// TIA Portal V20 export
TYPE "LConSMC_typePIDController"
// stored: Access Published
   STRUCT
      In { S7_SetPoint := 'True'} : "LConSMC_typePIDControllerIn";
      Out { S7_SetPoint := 'True'} : "LConSMC_typePIDControllerOut";
   END_STRUCT;
END_TYPE
